// TIA Portal V16 export
// export: Created 2021-11-12T13:32:57.4949609Z, ExportSetting WithDefaults, DisplayName Totally Integrated Automation Portal, DisplayVersion V16 Update 3, DisplayName TIA Portal Version Control Interface, DisplayVersion V16 Update 2, DisplayName TIA Portal Openness, DisplayVersion V16 Update 3, DisplayName SINAMICS Startdrive Advanced, DisplayVersion V16 Update 5, DisplayName SINAMICS Startdrive G130, G150, S120, S150, SINAMICS MV, S210, DisplayVersion V16 Update 5, DisplayName SINAMICS Startdrive G110M, G120, G120C, G120D, G120P, G115D, DisplayVersion V16 Update 5, DisplayName STEP 7 Professional, DisplayVersion V16 Update 3, DisplayName STEP 7 Safety, DisplayVersion V16, DisplayName WinCC UA Professional, DisplayVersion V16 Update 3
DATA_BLOCK "STATUS_Zone300"   // DB85
{ S7_Optimized_Access := 'TRUE'; DB_Accessible_From_OPC_UA := 'FALSE' }
VERSION : 0.1
// stored: AutoNumber true, DBAccessibleFromOPCUA false, IsOnlyStoredInLoadMemory false, IsRetainMemResEnabled false, IsWriteProtectedInAS false, MemoryReserve 100
   VAR
      Mode : Struct   // Statuses and error of zone 300
         Main : "UDT_Status_main";
         Specific : "UDT_Zone_Status_specific";
         Error : "UDT_Error01";
      END_STRUCT;
      StationBSN4_Mode : Struct   // Statuses and error of station BSN4
         Main : "UDT_Status_main";
         Specific : "UDT_Zone_Status_specific";
         Error : "UDT_Error01";
      END_STRUCT;
      StationBSN5_Mode : Struct   // Statuses and error of station BSN5
         Main : "UDT_Status_main";
         Specific : "UDT_Zone_Status_specific";
         Error : "UDT_Error01";
      END_STRUCT;
      Station310_Mode : Struct   // Statuses and error of station 310
         Main : "UDT_Status_main";
         Specific : "UDT_Zone_Status_specific";
         Error : "UDT_Error01";
      END_STRUCT;
      Station320_Mode : Struct   // Statuses and error of station 320
         Main : "UDT_Status_main";
         Specific : "UDT_Zone_Status_specific";
         Error : "UDT_Error01";
      END_STRUCT;
      Station330_Mode : Struct   // Statuses and error of station 330
         Main : "UDT_Status_main";
         Specific : "UDT_Zone_Status_specific";
         Error : "UDT_Error01";
      END_STRUCT;
   END_VAR
BEGIN
END_DATA_BLOCK
